{attribute 'GeneratedUsingTerminal: EL3611-1030-0016'}
{attribute addProperty BoxType "EL3611-1030-0016"}
{attribute addProperty Id "AI_InputsAT %I*AI_Inputs_4521310411WcStateAT %I*WcState_9091E0EB2InfoDataAT %I*InfoData_94A18F5E2"}
{attribute addProperty CRC "738885579"}
{attribute addProperty Size "15"}
TYPE EL3611_2C0A7FCB EXTENDS EtcSlaveTerminalBase_947E5A46 :
STRUCT
	{attribute addProperty Name "AI_Inputs"}
	AI_Inputs : AI_Inputs_45213104;
	{attribute addProperty Name "WcState"}
	WcState : WcState_9091E0EB;
	{attribute addProperty Name "InfoData"}
	InfoData : InfoData_94A18F5E;
END_STRUCT
END_TYPE

(* stored: Version 1.2.0.0, ProductVersion 3.1.4024.9
   DUT EL3611_2C0A7FCB: Id {69ce69e7-8c43-4929-9707-6ff70b2fb17d} *)
